PROGRAM SEQ_RW
VAR_INPUT
	RW_sequence	: UINT;
END_VAR

VAR
	process_X	: UINT; //Conveyor to Pitstop
	process_G	: UINT; //KR1 GET Magnet	
END_VAR


IF AUTO_MODE.KR1_PITSTOP THEN
	RETURN;
END_IF

CASE RW_sequence OF
	0:
		AUTO_MODE.processnameCR := CONCAT(MSG.COMP_RW,MSG.ACTION_INIT);	
		LOGPROCESS( spLogComp	 := MSG.COMP_RW, 
		 			spLogAction	 := MSG.ACTION_INIT, 
		 			spLogStatus	 := MSG.STATUS_DONE,
	 	 		 	plogFlag	 := TRUE);
		process_X	:= 0;
		process_G	:= 0;
		RW_sequence := 1;
		
	// Get Magnet -------------------------------------------------------------------------------------------------------------	
	1:
		IF NOT GVL.KR1_EOAT_FILL THEN
			IF process_G = 0 THEN
				IF KR1.Idle THEN
//					KR1.PLC_O_D3.0 := TRUE; //200
					KR1.bOutBit[3,0] := TRUE;
					AUTO_MODE.processnameCOSMO := CONCAT(MSG.COMP_RW,MSG.ACTION_GET_MAGNET);
					AUTO_MODE.processnameCOSMO := CONCAT(AUTO_MODE.processnameCOSMO,MSG.STATUS_RUN);
					LOGPROCESS( spLogComp	 := MSG.COMP_RW, 
								spLogAction	 := MSG.ACTION_GET_MAGNET, 
								spLogStatus	 := MSG.STATUS_RUN,
								plogFlag	 := TRUE);
					process_G := 1;
					RETURN;
				END_IF
			ELSIF process_G = 1 THEN
//				KR1.PLC_O_D3.0 := TRUE; //200
				KR1.bOutBit[3,0] := TRUE;
				IF NOT KR1.bInBit[3,0] THEN
//					KR1.PLC_O_D3.0 := FALSE; //200	
					KR1.bOutBit[3,0] := FALSE;
					AUTO_MODE.processnameCOSMO := CONCAT(MSG.COMP_RW,MSG.ACTION_GET_MAGNET);
					AUTO_MODE.processnameCOSMO := CONCAT(AUTO_MODE.processnameCOSMO,MSG.STATUS_ACK);
					LOGPROCESS( spLogComp	 := MSG.COMP_RW, 
								spLogAction	 := MSG.ACTION_GET_MAGNET, 
								spLogStatus	 := MSG.STATUS_ACK,
								plogFlag	 := TRUE);
					process_G := 2;
					RETURN;
				END_IF	
			ELSIF process_G = 2 THEN
//				KR1.PLC_O_D3.0 := FALSE; //200	
				KR1.bOutBit[3,0] := FALSE;
				IF KR1.bInBit[3,0] THEN
					AUTO_MODE.processnameCOSMO := CONCAT(MSG.COMP_RW,MSG.ACTION_GET_MAGNET);
					AUTO_MODE.processnameCOSMO := CONCAT(AUTO_MODE.processnameCOSMO,MSG.STATUS_DONE);
					LOGPROCESS( spLogComp	 := MSG.COMP_RW, 
								spLogAction	 := MSG.ACTION_GET_MAGNET, 
								spLogStatus	 := MSG.STATUS_DONE,
								plogFlag	 := TRUE);
					process_G:= 3;
					RETURN;
				END_IF	
			ELSIF process_G = 3 THEN
				IF KR1.Idle THEN
					AUTO_MODE.processnameCOSMO := CONCAT(MSG.COMP_RW,MSG.ACTION_GET_MAGNET);
					AUTO_MODE.processnameCOSMO := CONCAT(AUTO_MODE.processnameCOSMO,MSG.STATUS_COMP);
					LOGPROCESS( spLogComp	 := MSG.COMP_RW, 
								spLogAction	 := MSG.ACTION_GET_MAGNET, 
								spLogStatus	 := MSG.STATUS_COMP,
								plogFlag	 := TRUE);
					process_G := 4;
					RW_sequence := 2;
					AUTO_MODE.next_step := FALSE;
					GVL.KR1_EOAT_FILL := TRUE;
				END_IF
			END_IF
		ELSE
			RW_sequence := 2;
		END_IF
		
	// Conveyor to Pitstop -------------------------------------------------------------------------------------------------------------	
	2: 
		IF process_X = 0 THEN
			IF KR1.Idle AND NOT GVL.Rework_Empty THEN
//				KR1.PLC_O_D3.7 := TRUE; //206
				KR1.bOutBit[3,7] := TRUE;
				AUTO_MODE.processnameCOSMO := CONCAT(MSG.COMP_RW,MSG.ACTION_REWORK_IN);
				AUTO_MODE.processnameCOSMO := CONCAT(AUTO_MODE.processnameCOSMO,MSG.STATUS_RUN);
				LOGPROCESS( spLogComp	 := MSG.COMP_RW, 
							spLogAction	 := MSG.ACTION_REWORK_IN, 
							spLogStatus	 := MSG.STATUS_RUN,
							plogFlag	 := TRUE);
				process_X := 1;
				AUTO_MODE.RW_PACKING := TRUE;
				RETURN;
			END_IF
		ELSIF process_X = 1 THEN
//			KR1.PLC_O_D3.7 := TRUE; //206
			KR1.bOutBit[3,7] := TRUE;
			IF KR1.bInBit[3,7] THEN
//				KR1.PLC_O_D3.7 := FALSE; //206	
				KR1.bOutBit[3,7] := FALSE;
				AUTO_MODE.processnameCOSMO := CONCAT(MSG.COMP_RW,MSG.ACTION_REWORK_IN);
				AUTO_MODE.processnameCOSMO := CONCAT(AUTO_MODE.processnameCOSMO,MSG.STATUS_ACK);
				LOGPROCESS( spLogComp	 := MSG.COMP_RW, 
							spLogAction	 := MSG.ACTION_REWORK_IN, 
							spLogStatus	 := MSG.STATUS_ACK,
							plogFlag	 := TRUE);
				process_X := 2;
				RETURN;
			END_IF	
		ELSIF process_X = 2 THEN
//			KR1.PLC_O_D3.7 := FALSE; //206	
			KR1.bOutBit[3,7] := FALSE;
			IF NOT KR1.bInBit[3,7] THEN
				AUTO_MODE.processnameCOSMO := CONCAT(MSG.COMP_RW,MSG.ACTION_REWORK_IN);
				AUTO_MODE.processnameCOSMO := CONCAT(AUTO_MODE.processnameCOSMO,MSG.STATUS_DONE);
				LOGPROCESS( spLogComp	 := MSG.COMP_RW, 
							spLogAction	 := MSG.ACTION_REWORK_IN, 
							spLogStatus	 := MSG.STATUS_DONE,
							plogFlag	 := TRUE);
				process_X:= 3;
				RETURN;
			END_IF
		ELSIF process_X = 3 THEN
			IF KR1.Idle THEN
					AUTO_MODE.processnameCOSMO := CONCAT(MSG.COMP_RW,MSG.ACTION_REWORK_IN);
					AUTO_MODE.processnameCOSMO := CONCAT(AUTO_MODE.processnameCOSMO,MSG.STATUS_COMP);
					LOGPROCESS( spLogComp	 := MSG.COMP_RW, 
								spLogAction	 := MSG.ACTION_REWORK_IN, 
								spLogStatus	 := MSG.STATUS_COMP,
								plogFlag	 := TRUE);
					process_X := 4;
					RW_sequence := 3;
					AUTO_MODE.next_step := FALSE;
					AUTO_MODE.KR1_PITSTOP := TRUE;
				END_IF
		END_IF	
		
	3:
		RW_sequence := 0;
		AUTO_MODE.next_step := FALSE;
		AUTO_MODE.processnameRW := CONCAT(MSG.COMP_RW,MAIN.fb_TimeStamp.SystemTime);
		AUTO_MODE.processnameRW := CONCAT(AUTO_MODE.processnameRW,MSG.STATUS_END);
		LOGPROCESS( spLogComp	 := MSG.COMP_RW, 
					spLogAction	 := MSG.ACTION_REWORK_IN, 
					spLogStatus	 := MSG.STATUS_END,
					plogFlag	 := TRUE);
END_CASE

END_PROGRAM

(* stored: Version 1.1.0.1, ProductVersion 3.1.4024.12
   POU SEQ_RW: Id {1956c91f-91b4-46d5-bf62-e089dbee7ad6}, SpecialFunc None *)
